// TIA Portal project "Project1" (V16)

(* hardware
DEVICE "S7-1200 station_1"  S7-1200 Station
   slot 0: "Rack_0"  S7-1200 Rack  Rack  V1.0
DEVICE "S7-1200 station_3"  S7-1200 Station
   slot 0: "Rack_0"  S7-1200 Rack  Rack  V1.0
   slot 1: "ppppp"  CPU 1214C AC/DC/Rly  6ES7 214-1BG40-0XB0  V4.2
   slot 3: "AQ 1x12BIT_1"  AQ1 signal board  6ES7 232-4HA30-0XB0  V1.0
DEVICE "ET 200SP station_1"  ET 200SP-Station
   slot 0: "Rack_0"  Rack  6ES5 710-8MAx1
   slot 0: "robot"  IM 155-6 PN HF  6ES7 155-6AU00-0CN0  V3.3
   slot 1: "DI 8x24VDC HF_1"  DI 8x24VDC HF  6ES7 131-6BF00-0CA0  V2.0
      slot 1: "DI 8x24VDC HF_1"  DI 8x24VDC HF
   slot 2: "DI 8x24VDC HF_2"  DI 8x24VDC HF  6ES7 131-6BF00-0CA0  V2.0
      slot 1: "DI 8x24VDC HF_2"  DI 8x24VDC HF
   slot 3: "DQ 8x24VDC/0.5A HF_1"  DQ 8x24VDC/0.5A HF  6ES7 132-6BF00-0CA0  V2.0
      slot 1: "DQ 8x24VDC/0.5A HF_1"  DQ 8x24VDC/0.5A HF
   slot 4: "DQ 8x24VDC/0.5A HF_2"  DQ 8x24VDC/0.5A HF  6ES7 132-6BF00-0CA0  V2.0
      slot 1: "DQ 8x24VDC/0.5A HF_2"  DQ 8x24VDC/0.5A HF
   slot 5: "DI 8x24VDC HF_3"  DI 8x24VDC HF  6ES7 131-6BF00-0CA0  V2.0
      slot 1: "DI 8x24VDC HF_3"  DI 8x24VDC HF
   slot 6: "DQ 8x24VDC/0.5A HF_3"  DQ 8x24VDC/0.5A HF  6ES7 132-6BF00-0CA0  V2.0
      slot 1: "DQ 8x24VDC/0.5A HF_3"  DQ 8x24VDC/0.5A HF
   slot 7: "Server module_1"  Server module  6ES7 193-6PA00-0AA0  V1.1
      slot 1: "Server module_1"  Server module
   slot 127: "BA 2xRJ45"  BA 2xRJ45  6ES7 193-6AR00-0AA0  V0.0
      slot 1: "Port_1"  X1 P1 R  6ES7 193-6AR00-0AA0  V0.0
      slot 2: "Port_2"  X1 P2 R  6ES7 193-6AR00-0AA0  V0.0
DEVICE "HMI_1"  TP700 Comfort
   slot 0: "HMI_1"  TP700 Comfort  6AV2 124-0GC01-0AX0  14.0.1.0
   slot 1: "HMI_RT_1"  TP700 Comfort  6AV2 124-0GC01-0AX0  14.0.1.0
   slot 5: "HMI_1.IE_CP_1"  PROFINET Interface  14.0.1.0
      slot 1: "PROFINET Interface_1"  PROFINET Interface
         slot 1: "Port_1"  Port
         slot 2: "Port_2"  Port
   slot 7: "HMI_1.MPI/DP_CP_1"  MPI/DP Interface  14.0.1.0
*)

// ===== PLC "ppppp"  CPU 1214C AC/DC/Rly =====

VAR_GLOBAL   // PLC tag table "Variables_1"
   "Marcha" AT %I0.1 : Bool;
   "Paro" AT %I0.2 : Bool;
   "Habilitación" AT %M0.0 : Bool;
END_VAR

FUNCTION "Sección_1" : Void   // FC2, LAD
{ S7_Optimized_Access := 'TRUE' }
VERSION : 0.1
BEGIN

REGION Network 1
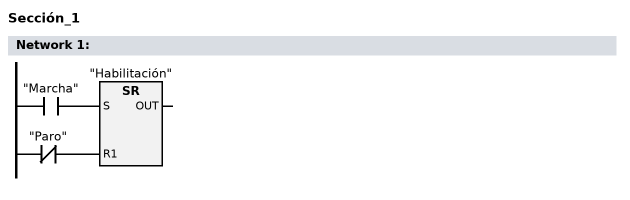
   RUNG wire#powerrail
      Contact( "Marcha" )
      S_SR(operand := "Habilitación", r1 := wire#w1)
   END_RUNG
   RUNG wire#powerrail
      I_Contact( "Paro" )
   END_RUNG wire#w1
   // the same network as SCL:
   IF "Marcha" THEN
       "Habilitación" := TRUE;   // SR flip-flop
   END_IF;
   IF NOT "Paro" THEN "Habilitación" := FALSE; END_IF;
END_REGION
END_FUNCTION

ORGANIZATION_BLOCK "Main"   // OB1, LAD, ProgramCycle
TITLE = "Main Program Sweep (Cycle)"
{ S7_Optimized_Access := 'TRUE' }
VERSION : 0.1
   VAR_INPUT
      Initial_Call : Bool;   // Initial call of this OB
      Remanence : Bool;   // =True, if remanent data are available
   END_VAR
BEGIN

REGION Network 1
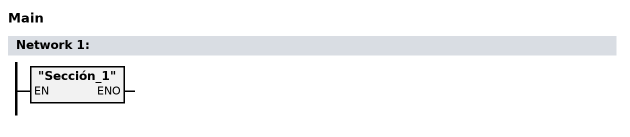
   RUNG wire#powerrail
      "Sección_1"()
   END_RUNG
   // the same network as SCL:
   "Sección_1"();
END_REGION
END_ORGANIZATION_BLOCK

(* ===== HMI "HMI_RT_1" =====
system functions are stored by id; their names below are inferred from use
connection "HMI_Connection_1": ETHERNET, S7_1200_OMS

HMI tags "Default tag table"
   "DB_HMI_Marcha" : Bool = PLC DB_HMI.Marcha, 1 s
   "DB_HMI_Paro" : Bool = PLC DB_HMI.Paro, 1 s
   "DB_HMI_En_marcha" : Bool = PLC DB_HMI.En_marcha, 1 s

screen "Root screen" 800x480, template "Template_1"
   Button "Button_1" at 25,147 size 96x32; TextOff 'Marcha'
      on Press: SetBit("DB_HMI_Marcha")
      on Release: ResetBit("DB_HMI_Marcha")
   Button "Button_2" at 25,204 size 96x32; TextOff 'Paro'
      on Press: SetBit("DB_HMI_Paro")
      on Release: ResetBit("DB_HMI_Paro")
   Circle "Circle_1" at 143,166 size 48x48
      Appearance <- "DB_HMI_En_marcha"
*)